Fanuc KAREL source: kc00030.KL

-- PROVISIONAL review KL for V770-1; original PC SHA256 7343bd6f478f36e52aa63340506f502015e1be6e9089faf9640b370dffde8f3b
-- Incomplete behavior may be omitted. Consult companion uncertainty JSON. Do not deploy.
PROGRAM KC00030
%NOLOCKGROUP
BEGIN
  -- UNRESOLVED_PC offsets 5-17; opcodes 3F,75
  -- UNRESOLVED_PC offsets 22-94; opcodes 27,22,2A,22,22,22,22,22,22,22,22,22,22,31
  -- UNRESOLVED_PC offsets 99-103; opcodes 7F
END KC00030
